(* CoDeSys 2.3 library: My_lib.lib *)
(* Libraries: C:\Program Files (x86)\WAGO Software\CODESYS V2.3\Targets\WAGO\Libraries\32_Bit\SysLibTime.lib 8.11.10 13:37:48, STANDARD.LIB 2.6.14 10:37:46 *)

(* Data type *)
TYPE AnalogScale :  (*параметры масштабирования аналоговых датчиков*)
STRUCT
	Block			: BOOL;	(*блокировка датчика и присвоение ему значения CurvalBlock - MW0.0*)
	Zero			: BOOL;	(*обнуление при масштабировании датчика уровня               	- MW0.8*)
	MaxKod    		: REAL;	(*макс код АЦП аналогового входа                                          	- MW2*)
	MinKod    		: REAL;	(*мин код АЦП аналогового входа                                           	- MW4*)
	MaxVal    		: REAL;	(*макс значение датчика в физических единицах                    - MW6*)
	MinVal    		: REAL;	(*мин значение датчика в физических единицах                      - MW8*)
	CurvalBlock		: REAL;	(*значение присваиваемое при блокировке датчика                - MW10*)
	Calibr       		: REAL;	(*значение калибровки показаний +-                                         	- MW12 *)
	ErrorLevel		: REAL; 	(*уровень помехи отклонения от усред величины для фильтрации  - MW14*)
	Hight_LE		: REAL;	(*высота танка, в метрах, при расчете уровня в %			- MW16*)
	NumbSample	: INT;       (*количество сэмплов для усреднения величины для фильтрации  - MW18*)
END_STRUCT
END_TYPE

(* Data type *)
TYPE START_UP_SI :
STRUCT
    EV_CLASS:   BYTE;
    EV_NUM:     BYTE;
    PRIORITY:   BYTE;
    NUM:        BYTE;
    TYP2_3:     BYTE;
    TYP1:       BYTE;
    ZI1:        WORD;
    ZI2_3:      DWORD;
END_STRUCT
END_TYPE

(* Data type *)
TYPE TOP_SI
 STRUCT
    EV_CLASS:   BYTE;
    EV_NUM:     BYTE;
    PRIORITY:   BYTE;
    NUM:        BYTE;
    TYP2_3:     BYTE;
    TYP1:       BYTE;
    ZI1:        WORD;
    ZI2_3:      DWORD;
END_STRUCT
END_TYPE

(* POU PLC_PRG, ST *)
PROGRAM PLC_PRG
	VAR_INPUT
	END_VAR
VAR

END_VAR
(* История изменений
26.03 - в AnalogSensor добавлена задержка времени срабатывания аварии датчика
12.07 - добавлен fb_AnScaling, объединяющий  Analog_Sensor и Filter,
  добавлена структура  AnalogScale - параметры масштабирования аналоговых датчиков.

*)
END_PROGRAM

(* POU Analog_Sensor, ST *)
FUNCTION_BLOCK Analog_Sensor
VAR_INPUT
	IsV: WORD;     (*значение на входе в модуль*)
	MaxKod: REAL;
	MinKod: REAL;
	MaxVal: REAL;
	MInVal: REAL;
	CurvalBlock: REAL;
	Calibr: REAL;
	HightTank: REAL; (*высота танка, для датчиков уровня*)
	SensorType: INT; (*тип датчика: 0-датчик уровня, 1-аналог 4-20 или 0-10, 3 - РТ100*)
	Block: BOOL;
	Time_DelayAlarm :TIME;  (*время задержки срабатывания аварии датчика*)
END_VAR
VAR_OUTPUT
	Error: BOOL;
	Result: REAL;
END_VAR
VAR
	Temp_IsV: REAL;
	T_Alarm: TON;  (*таймер срабатывания аварии датчика*)
END_VAR
(*обнуление*)
Result :=0.0;
T_Alarm.IN := FALSE;

CASE SensorType OF
0:(*для датчиков уровня 4-20мА*)
	IF ((IsV AND 16#0003) <> 16#0003) THEN  (*сравниваем с кодом ошибки входа*)
		Temp_IsV := WORD_TO_REAL(IsV);
  		Result := (Temp_IsV - MinKod) * ((MaxVal-MInVal)/(MaxKod-MInKod))+MInVal+Calibr;
	    	(*пересчет уровня в баках в %; HightTank - макс возможная высота столба в баке м, 10.197м - высота столба воды на 1 бар*)
  		Result := (Result*10.197)/HightTank*100;
	  	IF Result<0 THEN
    			Result:= 0.0;
	  	END_IF;
	ELSE                                 (*неисправность датчика или линии*)
		T_Alarm.IN := TRUE;
	END_IF;


1: (*для датчиков 4-20мА, 0-10В*)
	IF ((IsV AND 16#0003) <> 16#0003) THEN  (*сравниваем с кодом ошибки входа*)
  		Temp_IsV := WORD_TO_REAL(IsV);
	  	Result := (Temp_IsV - MinKod) * ((MaxVal-MInVal)/(MaxKod-MInKod))+MInVal+Calibr;
	ELSE                              (*неисправность датчика или линии*)
		T_Alarm.IN := TRUE;
	END_IF;

2:(* для РТ100*)
	Temp_IsV := WORD_TO_REAL(IsV);
	IF (Temp_IsV>-300) AND (Temp_IsV<1500) THEN
	  Result := Temp_IsV/10.0+Calibr;
	ELSE                            (*неисправность датчика или линии*)
		T_Alarm.IN := TRUE;
	END_IF;

END_CASE;

(*блокировка датчика с присвоением значений*)
IF Block THEN
   Result := CurvalBlock;
END_IF;

T_Alarm(PT:= Time_DelayAlarm, Q=>Error);  (*время задержки срабатывания аварии*)
END_FUNCTION_BLOCK

(* POU AnScaling, ST *)
FUNCTION_BLOCK AnScaling (*блок масштабирования и фильтрации аналоговых входов*)
VAR_INPUT
	i_IW_an       		:WORD; (*немасштабированный сигнал с физического входа*)
	i_SensorType	:INT;	(*тип датчика: 0 - уровень в танке 0..100%, 1 - аналоговый обычный, 2 - термосопротивление*)
END_VAR
VAR_OUTPUT
	q_Error         	: BOOL;  (*обшибка датчика*)
	q_LE    			: REAL;  (*масштабированное значение датчика*)
END_VAR
VAR
	fb_Sensor 	:Analog_Sensor;
	fb_Filtr 	:Filter;
END_VAR
VAR_IN_OUT
	i_An_Scale	: AnalogScale;	(*параметры масштабирования аналоговых датчиков*)
END_VAR
(*блок масштабирования*)
fb_Sensor(
	IsV:=			i_IW_an ,
	MaxKod:=		i_An_Scale.MaxKod ,
	MinKod:=		i_An_Scale.MinKod ,
	MaxVal:=		i_An_Scale.MaxVal ,
	MInVal:=			i_An_Scale.MinVal ,
	CurvalBlock:=	i_An_Scale.CurvalBlock ,
	Calibr:=			i_An_Scale.Calibr ,
	HightTank:=		i_An_Scale.Hight_LE ,
	SensorType:=	i_SensorType ,
	Block:=			i_An_Scale.Block ,
	Error=>			q_Error ,
	Result=>		fb_Filtr.Input );

(*блок фильтрации*)
fb_Filtr(
	MaxVal:=		i_An_Scale.MaxVal ,
	ErrorLevel:=		i_An_Scale.ErrorLevel ,
	NumbSample:=	i_An_Scale.NumbSample ,
	Result=>		q_LE );


IF i_An_Scale.Zero THEN           (*установка 0 датчика уровня*)
   	i_An_Scale.MinKod := fb_Sensor.IsV;
END_IF;
END_FUNCTION_BLOCK

(* POU Filter, ST *)
FUNCTION_BLOCK Filter
VAR_INPUT
	Input: REAL;  (*входное значение величины*)
	MaxVal: REAL; (* макс значение вход величины*)
	ErrorLevel: REAL;(*уровень помехи отклонения от сред величины*)
	NumbSample: INT; (*количество сэмплов для усреднения величины*)
END_VAR
VAR_OUTPUT
	Result:  REAL;
END_VAR
VAR
	Count: INT ;
	CountBadSample: INT; (*количество плохих сэмплов*)
	Sum: REAL;
END_VAR
 IF (((Result-Input)/MaxVal) < ErrorLevel AND ((Result-Input)/MaxVal) > (-ErrorLevel)) OR Input=0.0 OR Result=0.0  THEN
   Sum:=Input+Sum;
   CountBadSample:=0;
 ELSE
   Sum:=Result+Sum;
   CountBadSample:=CountBadSample+1;
 END_IF;


   IF Count>=NumbSample THEN
      Result:= Sum/NumbSample; (*результат - сумма замеров / на кол-во сэмплов*)
      Count:=1;
      Sum:=0.0;
   ELSE
      Count:=Count+1;
   END_IF;

   IF CountBadSample>(NumbSample*3) THEN (*если вышли за пределы и остались там*)
      Result:=Input;
      Sum:=0.0;
      Count:=1;
   END_IF;
END_FUNCTION_BLOCK

(* POU PID_M, ST *)
FUNCTION_BLOCK PID_M
VAR_INPUT
	i_DpartOff: BOOL := TRUE;
	i_PpartOff: BOOL:= FALSE;
	i_IpartOff: BOOL:= FALSE;
	i_Sp: REAL;
	i_PVin: REAL;
	i_Gain: REAL;
	i_Ti: REAL;
	i_Td: REAL;
	i_Max_Ipart: REAL;     (*ограничение интегральной составляющей регулятора*)
	i_Reset: BOOL:= FALSE;
	i_scan_time: REAL;
END_VAR
VAR_OUTPUT
	q_Err: BOOL;
	q_PV: REAL;
END_VAR
VAR
	Ppart: REAL;
	Ipart: REAL;
	Dpart: REAL;
	E: REAL;
	Esum: REAL;
	dE: REAL;
	Ep: REAL;
END_VAR
IF (i_Ti > 0.0) OR (i_scan_time >= 0.0) OR (i_Gain >= 0.0)
             OR ((i_SP >= 0.0) AND (i_SP <= 100.0))
             OR ((i_PVin >= 0.0) AND (i_PVin <= 100.0)) THEN
        E := i_Sp - i_PVin ;                                    (*значения в % от макс величины*)
        dE := E - Ep ;
        Esum := Esum + E * i_scan_time ;

        IF NOT i_PpartOff THEN
            Ppart := i_Gain * E ;
        ELSE
            Ppart := 0.0 ;
        END_IF;

        IF NOT i_IpartOff THEN
           Ipart := Esum / (i_Ti * 1000.0) ;
            IF Ipart>i_Max_Ipart THEN
               Esum := i_Max_Ipart * (i_Ti * 1000.0) ;
            ELSIF Ipart<=0 THEN
               Esum :=0.0;
             END_IF;
        ELSE
            Ipart := 0.0 ;
        END_IF;


        IF NOT i_DpartOff THEN
            Dpart := (i_Td * dE * 1000.0) /i_scan_time ;
        ELSE
            Dpart := 0.0 ;
        END_IF;

        q_PV := Ppart + Ipart + Dpart ;

        IF q_PV < 0.0 THEN
            q_PV := 0.0 ;
            (*Esum:=0;*)
        ELSIF q_PV > 100.0 THEN
            q_PV := 100.0 ;
        END_IF;

        q_Err := FALSE ;
    ELSE
        q_PV := 0.0 ;
        q_Err := TRUE ;
    END_IF;

    IF i_Reset THEN
        q_PV := 0.0 ;
        Esum := 0.0 ;
        Ipart :=0.0 ;
    END_IF;

    Ep := E ;
END_FUNCTION_BLOCK

(* POU Pump, ST *)
FUNCTION_BLOCK Pump
VAR_INPUT
	i_AlarmReset: BOOL; (*сброс аварии*)
	IsV_P: BOOL;        (*подтверждение включения*)
	Protect: BOOL;       (*защита двигателя*)
	SetV_P: BOOL;     (*команда на включение*)
	Timer_PT: TIME;    (*время таймера*)
END_VAR
VAR_OUTPUT
	Alarm: BOOL;   (*авария *)
	q_P: BOOL;
END_VAR
VAR
	Mode: INT;
	T_VA : TON ;
END_VAR
 T_VA.PT:=Timer_PT;
 q_P := FALSE;
 Alarm :=FALSE;

CASE Mode OF
0: (*выключен *)
   T_VA.IN :=  IsV_P  ;
   IF T_VA.Q OR Protect THEN
      T_VA.IN := FALSE;
      Mode:=2;
   END_IF;
  IF SetV_P THEN
     Mode:=1;
   END_IF;


 1: (*запущен*)
    T_VA.IN :=NOT IsV_P ;
    IF T_VA.Q OR Protect THEN
      T_VA.IN := FALSE;
      Mode:=2;
   END_IF;
  IF NOT SetV_P THEN
     Mode:=0;
  END_IF;
  q_P := TRUE;

 2: (* авария *)
    Alarm :=TRUE;
    IF i_AlarmReset AND NOT Protect THEN
       Mode:=0;
     END_IF;
END_CASE;

T_VA();
END_FUNCTION_BLOCK

(* POU TimerIncr, ST *)
FUNCTION_BLOCK TimerIncr (*Расчет времени скана*)
VAR_INPUT
END_VAR
VAR_OUTPUT
	q_scan_time: REAL;
END_VAR
VAR
 Cur_Time    : DWORD ;       (*Текущее время*)
 PastTime   : DWORD;       (*Время на предыдущем скане*)
 Sys_Time: SysTime64;
 CurrentTime:CurTime;  (*блок определения систем времени*)
END_VAR
Sys_time.ulHigh :=0; (*обнуление*)
Sys_time.ulLow :=0;
CurrentTime(SystemTime:= Sys_Time);
Cur_Time := Sys_time.ulLow;
q_scan_time:=(DWORD_TO_REAL(Cur_Time-PastTime)/1000.0); (*получение текущего системного времени в мс*)
PastTime := Cur_Time;
END_FUNCTION_BLOCK

(* POU Valve, ST *)
FUNCTION_BLOCK Valve
VAR_INPUT
	i_AlarmReset: BOOL; (*сброс аварии*)
	i_VAopen: BOOL;        (*датчик положения - клапан открыт*)
	i_VAclose: BOOL;        (*датчик положения - клапан закрыт*)
	i_DiagVA: BOOL;       (*вклюечение диагностики клапана*)
	i_SetVA: BOOL;     (*команда на включение*)
	i_TimerPT: TIME;    (*время таймера*)
END_VAR
VAR_OUTPUT
	q_Alarm: BOOL;   (*авария клапана*)
	q_VA: BOOL;
END_VAR
VAR
	Mode: INT;
	T_VA : TON ;
END_VAR
 T_VA.PT:=i_TimerPT;
 q_VA := FALSE;
 q_Alarm :=FALSE;

CASE Mode OF
0: (*клапан закрыт (по умолчанию) *)
   T_VA.IN := NOT i_VAclose AND i_DiagVA; (*если нет сигнала с датчика и включена диагностика*)
   IF T_VA.Q THEN
      T_VA.IN := FALSE;
      Mode:=2;
   END_IF;
  IF i_SetVA THEN  (*если подали сигнал то на открытие*)
     Mode:=1;
   END_IF;


 1: (*клапан открыт*)
    T_VA.IN :=NOT i_VAopen AND i_DiagVA; (*если сигнал с датчика остался и включена диагностика*)
    IF T_VA.Q THEN
      T_VA.IN := FALSE;
      Mode:=2;
   END_IF;
  IF NOT i_SetVA THEN (*если сняли сигнал то на закрытие*)
     Mode:=0;
  END_IF;
  q_VA := TRUE;

 2: (* авария клапана*)
    q_Alarm :=TRUE;
    IF i_AlarmReset THEN
       Mode:=0;
     END_IF;
END_CASE;

T_VA();
END_FUNCTION_BLOCK
